// TwinCAT 3 PLC project RpcServer
// ProgramVersion: 3.1.4024.0
// libraries:
//   rplc, * (tchaxx)
//   Tc2_Standard, * (Beckhoff Automation GmbH)
//   Tc2_System, * (Beckhoff Automation GmbH)
//   Tc3_Module, * (Beckhoff Automation GmbH)
// project tree:
//   DUTs/ ST_Subscriber.TcDUT
//   / PlcTask.TcTTO
//   POUs/ FB_Publisher.TcPOU, FB_RpcServer.TcPOU, MAIN.TcPOU

CONFIGURATION RpcServer
    RESOURCE PLC ON TwinCAT3
        TASK PlcTask(INTERVAL := T#10ms, PRIORITY := 21);
        PROGRAM MAIN WITH PlcTask : MAIN;
    END_RESOURCE
END_CONFIGURATION

// ---- DUTs/ST_Subscriber.TcDUT
TYPE ST_Subscriber :
STRUCT
	nHandle			: UDINT;
	stAdsStatus		: ST_AdsStatus;
	fbRPC			: FB_RPC_Dynamic;
END_STRUCT
END_TYPE

// ---- POUs/MAIN.TcPOU
PROGRAM MAIN
VAR
	{attribute 'analysis' := '-33'}
	fbRpcServer : FB_RpcServer;
	
	fbPublisher	: FB_Publisher;		// PubSub example
END_VAR


fbPublisher();

END_PROGRAM

// ---- POUs/FB_RpcServer.TcPOU
FUNCTION_BLOCK FB_RpcServer
VAR_INPUT
END_VAR
VAR_OUTPUT
END_VAR
VAR
END_VAR

{attribute 'TcRpcEnable'}
METHOD Greet : T_MaxString
VAR_INPUT
	sName : T_MaxString;
END_VAR
VAR_OUTPUT
	nLen : INT;
END_VAR
VAR_IN_OUT CONSTANT
	stLibVersion : ST_LibVersion;
END_VAR

Greet := CONCAT(CONCAT(CONCAT('Hello ', sName), '! LibVersion: '), stLibVersion.sVersion);

nLen := LEN(Greet);
END_METHOD

END_FUNCTION_BLOCK

// ---- POUs/FB_Publisher.TcPOU
FUNCTION_BLOCK FINAL FB_Publisher

VAR
	aSubscribers	: ARRAY[0..cSubsUpperBound] OF ST_Subscriber;	
END_VAR

VAR_TEMP
	nTrigger		: UDINT;
END_VAR

VAR CONSTANT
	cSubsUpperBound	: UDINT := 9;
	cTrigger		: UDINT := 50;
END_VAR

nTrigger := _TaskInfo[GETCURTASKINDEXEX()].CycleCount MOD cTrigger;
IF nTrigger = 0 THEN
	InvokeSubscribersCallback(_TaskInfo[GETCURTASKINDEXEX()].CycleCount);
END_IF

InvokeSubscriberWhileBusy();

METHOD PRIVATE InvokeSubscribersCallback
VAR_INPUT
	nTrigger : UDINT;
END_VAR

VAR
	i 	: UDINT;
	refSub : REFERENCE TO ST_Subscriber;
END_VAR

FOR i:= 0 TO cSubsUpperBound DO
	refSub REF= aSubscribers[i];
	
	IF refSub.nHandle = 0 THEN
		CONTINUE;
	END_IF
	
	refSub.stAdsStatus := refSub.fbRPC.VarInput(nTrigger).NoReturnValue().Invoke();

END_FOR
END_METHOD

METHOD PRIVATE InvokeSubscriberWhileBusy

VAR
	i 		: UDINT;
	refSub : REFERENCE TO ST_Subscriber;
END_VAR

FOR i:= 0 TO cSubsUpperBound DO
	
	refSub REF= aSubscribers[i];
	IF refSub.nHandle = 0 OR_ELSE NOT refSub.stAdsStatus.bBusy THEN
		CONTINUE;
	END_IF
	
	refSub.stAdsStatus := refSub.fbRPC.Invoke();

END_FOR
END_METHOD

{attribute 'TcRpcEnable'}
METHOD PRIVATE Subscribe : HRESULT
VAR_INPUT CONSTANT
	sAmsNetId		: T_AmsNetID;
	nPort			: T_AmsPort;
	sInstancePath	: STRING;
	sSymbol			: STRING;
END_VAR
VAR_OUTPUT
	nHandle : UDINT;
END_VAR

VAR 
	i	: UDINT;
END_VAR

VAR_INST
	nHandleCnt			: UDINT;
	fbCrititcalSection 	: FB_IecCriticalSection;
END_VAR
Subscribe := S_PENDING;

(* start of critical section *)
IF fbCrititcalSection.Enter() THEN
    
	FOR i := 0 TO cSubsUpperBound DO	
		IF aSubscribers[i].nHandle > 0 THEN
			CONTINUE;
		END_IF
		nHandleCnt := nHandleCnt + 1;
		aSubscribers[i].nHandle := nHandleCnt;		
		aSubscribers[i].fbRPC.Configure().WithAmsNetId(sAmsNetId).WithAmsPort(nPort).WithSymbolPath(sInstancePath, sSymbol).Build();
		nHandle := nHandleCnt;
		Subscribe := S_OK;
		EXIT;
	END_FOR
	
    (* end of critical section *)
	fbCrititcalSection.Leave();
END_IF
END_METHOD

{attribute 'TcRpcEnable'}
METHOD PRIVATE Unsubscribe : HRESULT
VAR_INPUT
	nHandle	: UDINT;
END_VAR

VAR 
	i		: UDINT;
	refSub 	: REFERENCE TO ST_Subscriber;
END_VAR

VAR_INST
	fbCrititcalSection 	: FB_IecCriticalSection;
END_VAR
Unsubscribe := S_FALSE;

(* start of critical section *)
IF fbCrititcalSection.Enter() THEN
    
	FOR i := 0 TO cSubsUpperBound DO
		
		refSub REF= aSubscribers[i];	
		IF refSub.nHandle = 0 OR_ELSE refSub.nHandle <> nHandle THEN
			CONTINUE;
		END_IF
		
		refSub.nHandle := 0;	
		Unsubscribe := S_OK;
		EXIT;
	END_FOR
	
    (* end of critical section *)
	fbCrititcalSection.Leave();
END_IF
END_METHOD

END_FUNCTION_BLOCK
